TYPE DS_BrensonMulFreqSwitching :
STRUCT
	bFreqSwitchingPB_TS : BOOL;
	bFreqRange4080120En : BOOL;
	bFreqRange2550En : BOOL;
	bDisableMultiFreq80kHz : BOOL;
	iFreqOutput_TS : INT;
END_STRUCT
END_TYPE

(* stored: Version 1.1.0.1, ProductVersion 3.1.4024.12
   DUT DS_BrensonMulFreqSwitching: Id {b4219dfb-2cfb-44c7-bc81-966e8c5f78a0} *)
